FUNCTION_BLOCK FB_WorkerDefGrid_Inspection EXTENDS FB_WorkerDefGrid
VAR PERSISTENT
  _fWorkerToMasterRef  : LREAL := 3;    (*Distance between Master reference first PM and this worker, mechanisch*)
END_VAR


{warning 'TODO: implement inspection trigger'}

METHOD PROTECTED  Attach : BOOL
VAR_INPUT
  iCT              : I_CT;                         (*container at triggered event position*)
END_VAR
IF SUPER^.Attach(iCT:=iCT) THEN
  ;
END_IF
END_METHOD

PROPERTY fWorkerToMasterRef : LREAL
GET
fWorkerToMasterRef := _fWorkerToMasterRef;
END_GET
END_PROPERTY

METHOD   mJobStart
VAR_INPUT
	sJobDef	: CalmarCompPrint.I_JobDefinition;
END_VAR
END_METHOD

METHOD  mJobStop
VAR_INPUT
	sStatus	: CalmarCompPrint.I_JobStatus;
END_VAR
END_METHOD

METHOD Release : BOOL
VAR_INPUT
  iCT              : I_CT;                         (*container at triggered event position*)
END_VAR
IF SUPER^.Release(iCT := iCT) THEN
  ;  
END_IF
END_METHOD

METHOD  work
SUPER^.work();

//Worker position update
IF _iWorkerParams <> 0 AND _pAttachedCt = 0 THEN     // Update only without attached container
  // WorkerPosition =  Worker<-Master<-CAM<-SheetDetect
  fPosition := _fWorkerToMasterRef + _iWorkerParams.fDetectToRefPos;
END_IF

IF _pAttachedCt <> 0 THEN
  Release(iCT:=_pAttachedCt^);
END_IF
END_METHOD

END_FUNCTION_BLOCK

(* stored: Version 1.1.0.1, ProductVersion 3.1.4024.11
   POU FB_WorkerDefGrid_Inspection: Id {37a97a00-485c-4f31-b7d7-7fb45a0dff8b}, SpecialFunc None
   Folder I_PrintStatusClient: Id {f1eb16b3-4bb7-4cf8-afe5-945958c7b424}
   Method Attach: Id {dd02a3c2-da79-4b50-92d0-e58ec36803fd}
   Property fWorkerToMasterRef: Id {d58f24b0-0176-4ca2-917c-0b196b6c3f32}
   Get Get: Id {1eaedd67-6f89-4513-9eb9-7f355cc38bbe}
   Method mJobStart: Id {3edbf743-26ae-401c-b89d-f5fce7aeb73d}
   Method mJobStop: Id {2fd18750-e428-4c8f-8165-dc217acd925e}
   Method Release: Id {e32eff20-e77d-40b3-9c81-5ebcb6e13ebd}
   Method work: Id {d1975cf7-7637-4f43-beac-caa62ff485b7} *)
